// :Description: Example interface for TcKit parser validation.
INTERFACE I_Example


// :Description: Execute one cycle.
// :returns: TRUE when the operation completes
METHOD Execute : BOOL
VAR_INPUT
    bTrigger : BOOL;
END_VAR
END_METHOD


// :Description: Reset to idle state.
// :returns: TRUE on success
METHOD Reset : BOOL
END_METHOD


// :Description: Current status word.
PROPERTY Status : DWORD
GET
END_GET
END_PROPERTY

END_INTERFACE

(* stored: Version 1.1.0.1, ProductVersion 3.1.4026.0
   Itf I_Example: Id {12345678-0000-0000-0000-000000000020}
   Method Execute: Id {12345678-0000-0000-0000-000000000021}
   Method Reset: Id {12345678-0000-0000-0000-000000000022}
   Property Status: Id {12345678-0000-0000-0000-000000000023}
   Get: Id {12345678-0000-0000-0000-000000000024} *)
